{attribute 'qualified_only'}
{attribute 'strict'}
TYPE E_Msg_Acknowledge :
(
	ByOperator := 0,
	Auto := 1
)UINT;
END_TYPE

(* stored: Version 1.1.0.1, ProductVersion 3.1.4024.10
   DUT E_Msg_Acknowledge: Id {75bceae6-7a88-4327-bc31-c2ae049edcb2} *)
